FUNCTION F_TB_PV2REAL : REAL
VAR_INPUT
	PvStr: STRING;
END_VAR
VAR
	iPV: LINT;
	r1: REAL;
END_VAR

// SMC HEBC002-WA10
// sv >= 0 -> '00010'
// sv < 0 -> '-0010'
iPV := STRING_TO_LINT(PvStr);
r1 := LINT_TO_REAL(iPV);
F_TB_PV2REAL := r1 / 10;

END_FUNCTION

(* stored: Version 1.1.0.1, ProductVersion 3.1.4024.12
   POU F_TB_PV2REAL: Id {29079dae-059e-4bd8-b200-2aef2ca876c4}, SpecialFunc None *)
